// TIA Portal V18 export
DATA_BLOCK "07_DOOR"   // DB48, F_DB
{ S7_Optimized_Access := 'TRUE'; DB_Accessible_From_OPC_UA := 'FALSE' }
// stored: DBAccessibleFromOPCUA false
   VAR
      AlwaysFALSE : Bool;
      AlwaysTRUE : Bool := TRUE;
      "!!ITERATOR_STRINGS$$" : Bool;
      "!!07_DOOR.{db_element:DI1/2}$$" : Bool;
      "!!07_DOOR.{db_element:DI2/2}$$" : Bool;
      "!!07_DOOR.{db_element:DD}$$" : Bool;
   END_VAR
BEGIN
END_DATA_BLOCK
